// TIA Portal V17 export
// export: Created 2021-12-03T08:08:03.8089922Z, ExportSetting WithDefaults, DisplayName Totally Integrated Automation Portal, DisplayVersion V17, DisplayName TIA Portal Openness, DisplayVersion V17, DisplayName TIA Portal Version Control Interface, DisplayVersion V17, DisplayName STEP 7 Professional, DisplayVersion V17, DisplayName STEP 7 Safety, DisplayVersion V17, DisplayName WinCC Advanced, DisplayVersion V17
VAR_GLOBAL   // PLC tag table "Digital_Outputs"
   O_PrDoor1Lamp AT %Q0.0 : Bool;   // Protecting Door 1 Lamp
   O_PrDoor2Lamp AT %Q0.1 : Bool;   // Protecting Door 2 Lamp
   O_Spare0_2 AT %Q0.2 : Bool;   // Spare
   O_Spare0_3 AT %Q0.3 : Bool;   // Spare
   O_P3AckInSAreaLamp AT %Q0.4 : Bool;   // Panel 3: Acknowledgement in the Safety Area Lamp
   O_Spare0_5 AT %Q0.5 : Bool;   // Spare
   O_Spare0_6 AT %Q0.6 : Bool;   // Spare
   O_Spare0_7 AT %Q0.7 : Bool;   // Spare
   O_P1AckEmStpOutSAreaLamp AT %Q1.0 : Bool;   // Panel 1: Acknowledgement Emergency Stop outsite the Safety Area Lamp
   O_Spare1_1 AT %Q1.1 : Bool;   // Spare
   O_ChilVlvAcc1 AT %Q1.2 : Bool;   // Accelerator 1 chiller valve
   O_ChilVlvAcc2 AT %Q1.3 : Bool;   // Accelerator 2 chiller valve
   O_P2ConvFwd AT %Q1.4 : Bool;   // Panel 2: Conveyor move forward
   O_P2ConvBwd AT %Q1.5 : Bool;   // Panel 2: Conveyor move backward
   O_ModSwchAcc1 AT %Q1.6 : Bool;   // Accelerator 1 modulator switch
   O_ModSwchAcc2 AT %Q1.7 : Bool;   // Accelerator 2 modulator switch
   O_AccReqWarmUp AT %Q2.0 : Bool;   // Accelerator Request: Warming up
   O_AccReqXRayOn AT %Q2.1 : Bool;   // Accelerator Request: X-Ray on
   O_AccReqXRayNotOn AT %Q2.2 : Bool;   // Accelerator Request: X-Ray not on
   O_AccReqResetFlt AT %Q2.3 : Bool;   // Accelerator Request: Reset Fault
   O_AccReqWarmUpFull AT %Q2.4 : Bool;   // Accelerator Request: Warming up Full (Standby-Clear)
   O_AccReqMicroWaveOn AT %Q2.5 : Bool;   // Accelerator Request: Microwave on
   O_AccReqHighDozeOn AT %Q2.6 : Bool;   // Accelerator Request: HighDoze on
   O_StateSig1RedL AT %Q3.0 : Bool;   // State Signal 1: Red Light
   O_StateSig1YellowL AT %Q3.1 : Bool;   // State Signal 1: Yellow Light
   O_StateSig1GreenL AT %Q3.2 : Bool;   // State Signal 1: Green Light
   O_StateSig1Horn AT %Q3.3 : Bool;   // State Signal 1: Horn
   O_StateSig2WhiteL AT %Q3.4 : Bool;   // State Signal 2: White Light (X-Ray is ON)
   O_StateSig2Horn AT %Q3.7 : Bool;   // State Signal 2: Horn (X-Ray Starts)
   O_Spare2_7 AT %Q2.7 : Bool;   // Spare
   O_Spare3_5 AT %Q3.5 : Bool;   // Spare
   O_Spare3_6 AT %Q3.6 : Bool;   // Spare
END_VAR
